# EPICS substitutions: ek9000App/Db/EL3058.substitutions
file EL3058.template
{       pattern
        {
                TERMINAL,

        }
        {
        }
}
